FUNCTION FB_LowpassFilter : REAL;
VAR_INPUT
	rValueIn	:REAL;
END_VAR
VAR
	rValue_In	:REAL;
	rValue_New	:REAL;	
	rValue_Old	:REAL;
	rFactor	    :REAL := 0.1; // 10% old new value			

END_VAR

//***********************************************************************************
//
// 
// ***********************************************************************************
// 
// PROJECT     :  A061 
// 
// FUNCTION    :  
// 
// AUTHOR      :  Weiting Chen
// 
// EMAIL       :  
// 
// Copyright   :  
//
// ***********************************************************************************

//

rValue_In := rValueIn;

IF rValue_Old = 0 THEN;
	rValue_Old := rValue_In;
	rValue_New := ((1-rFactor)*rValue_Old) + (rFactor*rValue_In);
ELSE
	rValue_Old := rValue_New;
	rValue_New := ((1-rFactor)*rValue_Old) + (rFactor*rValue_In);
END_IF


// Read IO in and out
FB_LowpassFilter := rValue_New;

END_FUNCTION

(* stored: Version 1.1.0.1, ProductVersion 3.1.4024.2
   POU FB_LowpassFilter: Id {5fd9c30e-7d37-4f71-b563-ad00f4d23a52}, SpecialFunc None *)
